Fanuc KAREL source: ko00100.KL

-- PROVISIONAL review KL for V1013-1; original PC SHA256 bb3c2f70d93fd052c53c9889ad0f724bd13039b3deb0c6112920f353c0a884be
-- Incomplete behavior may be omitted. Consult companion uncertainty JSON. Do not deploy.
PROGRAM KO00100
%NOLOCKGROUP
VAR
  A : INTEGER
  B : REAL
  OUT : REAL
BEGIN
  -- UNRESOLVED_PC offsets 5-12; opcodes 9D,23
  -- UNRESOLVED_PC offsets 17-29; opcodes 2E,64,23
  -- UNRESOLVED_PC offsets 34-57; opcodes 27,27,21,64,22,76,23
  -- UNRESOLVED_PC offsets 62-66; opcodes 7F
END KO00100
